FUNCTION_BLOCK FB_LOG_Handler
VAR_INPUT
	_IsUsed					: BOOL;
	bLogData					: BOOL;
	sLogMessage				: T_LongSTRING;
END_VAR
VAR_IN_OUT
	stEventData				: ST_LOG_EventData;
END_VAR
VAR_OUTPUT
	bDone						: BOOL;
	bBufferOverflow			: BOOL;
END_VAR
VAR
	rtExecute					: R_TRIG;
	sString 					: T_LongSTRING;
	nStringLen					: UINT;

END_VAR

_IsUsed := TRUE;

rtExecute(CLK:=bLogData);

IF NOT stEventData.bBufferOverflow AND stEventData.bEnable AND sLogMessage <> '' AND rtExecute.Q THEN

	sString := '';
	(*stEventData.nCounter := stEventData.nCounter + 1;
	sString := F_CONCAT4(F_AddPaddingUDINT(stEventData.nCounter, 7), ' : ', stEventData.sTimeStamp, ' : ');*)
	//sString := CONCAT(stEventData.sTimeStamp, ' : ');
	//sString := F_LongCONCAT(sString,sLogMessage);
	//sString := F_LongCONCAT(sString,'.$R$N');
	CONCAT2(ADR(stEventData.sTimeStamp), ADR(' : '), ADR(sString), SIZEOF(sString));
	CONCAT2(ADR(sString), ADR(sLogMessage), ADR(sString), SIZEOF(sString));
	CONCAT2(ADR(sString), ADR('.$R$N'), ADR(sString), SIZEOF(sString));
	nStringLen := TO_UINT(LEN2(ADR(sString)));  //Max size 1024 byte -> LongString

	stEventData.nControlSize := stEventData.nControlSize + nStringLen;

	IF stEventData.nControlSize <  stEventData.nMaxImageArraySize THEN
		MEMMOVE(ADR(stEventData.aDataLogImage[stEventData.nImageByte]), ADR(sString), nStringLen);
		stEventData.nImageByte := stEventData.nImageByte + nStringLen;
	ELSE
		stEventData.bBufferOverflow	:=TRUE;
		bBufferOverflow	:= TRUE;
	END_IF

	bDone	:= TRUE;
	(*F_LOG_Handler := TRUE;*)
ELSE
	bDone	:= FALSE;
END_IF

END_FUNCTION_BLOCK

(* stored: Version 1.1.0.1
   POU FB_LOG_Handler: Id {e27b869d-ed7f-47b8-b920-0c00fdc051f4}, SpecialFunc None *)
